FUNCTION InfluxAddData_10Hz : BOOL
VAR_IN_OUT
	Data			: ST_DATA;
	DataCollector	: FB_InfluxDataCollector;
END_VAR

// =================== Example:
	DataCollector.AddLreal(	'Test',                      Data.Gps.Inputs.x);

END_FUNCTION

(* stored: Version 1.1.0.1, ProductVersion 3.1.4022.11
   POU InfluxAddData_10Hz: Id {dbd45c9a-931e-e7d9-c709-f37398582a5e}, SpecialFunc None *)
